TYPE WCHAR : WSTRING(1); END_TYPE

(* stored: Version 1.1.0.1, ProductVersion 3.1.4024.11
   DUT WCHAR: Id {78a33f81-04f7-4e26-abc3-9c3e15255ebe} *)
